// TIA Portal V16 export
// export: Created 2021-11-12T13:31:11.1513233Z, ExportSetting WithDefaults, DisplayName Totally Integrated Automation Portal, DisplayVersion V16 Update 3, DisplayName TIA Portal Version Control Interface, DisplayVersion V16 Update 2, DisplayName TIA Portal Openness, DisplayVersion V16 Update 3, DisplayName SINAMICS Startdrive Advanced, DisplayVersion V16 Update 5, DisplayName SINAMICS Startdrive G130, G150, S120, S150, SINAMICS MV, S210, DisplayVersion V16 Update 5, DisplayName SINAMICS Startdrive G110M, G120, G120C, G120D, G120P, G115D, DisplayVersion V16 Update 5, DisplayName STEP 7 Professional, DisplayVersion V16 Update 3, DisplayName STEP 7 Safety, DisplayVersion V16, DisplayName WinCC UA Professional, DisplayVersion V16 Update 3
DATA_BLOCK "IDB_Sfty_Input"   // DB181, F_DB
{ DB_Accessible_From_OPC_UA := 'FALSE' }
VERSION : 0.1
// stored: AutoNumber true, DBAccessibleFromOPCUA false, InstanceOfName Sfty_Input, InstanceOfType FB
"Sfty_Input"
   // VAR
   //    SF_KAS1 { S7_SetPoint := 'True'} : ESTOP1;
   //    SF_KAS2 { S7_SetPoint := 'True'} : ESTOP1;
   //    SF_BSN1_2 { S7_SetPoint := 'True'} : ESTOP1;
   //    SF_SCH1 { S7_SetPoint := 'True'} : ESTOP1;
   //    SF_BSN3 { S7_SetPoint := 'True'} : ESTOP1;
   //    SF_BSN4_5 { S7_SetPoint := 'True'} : ESTOP1;
   //    SF_THM1 { S7_SetPoint := 'True'} : ESTOP1;
   //    SF_THM2 { S7_SetPoint := 'True'} : ESTOP1;
   //    "SF_1R1-RC01" { S7_SetPoint := 'True'} : ESTOP1;
   //    "SF_1R2-RC01" { S7_SetPoint := 'True'} : ESTOP1;
   //    "SF_1R3-RC01" { S7_SetPoint := 'True'} : ESTOP1;
   //    "SF_1R4-RC01" { S7_SetPoint := 'True'} : ESTOP1;
   //    "SF_1R5-RC01" { S7_SetPoint := 'True'} : ESTOP1;
   //    "SF_1R6-RC01" { S7_SetPoint := 'True'} : ESTOP1;
   //    "SF_2R1-RC01" { S7_SetPoint := 'True'} : ESTOP1;
   //    "SF_2R2-RC01" { S7_SetPoint := 'True'} : ESTOP1;
   //    "SF_000UH11-SF01_12" { S7_SetPoint := 'True'} : ESTOP1;
   //    "SF_000UH10-SF01_12" { S7_SetPoint := 'True'} : ESTOP1;
   //    "SF_100UH11-SF01_12" { S7_SetPoint := 'True'} : ESTOP1;
   //    "SF_100UH12-SF01_12" { S7_SetPoint := 'True'} : ESTOP1;
   //    "SF_100UH13-SF01_12" { S7_SetPoint := 'True'} : ESTOP1;
   //    "SF_100UF01-SF01_12" { S7_SetPoint := 'True'} : ESTOP1;
   //    "SF_200UH11-SF01_12" { S7_SetPoint := 'True'} : ESTOP1;
   //    "SF_200UF01-SF01_12" { S7_SetPoint := 'True'} : ESTOP1;
   //    "SF_210UF01-SF01_12" { S7_SetPoint := 'True'} : ESTOP1;
   //    "SF_220UF01-SF01_12" { S7_SetPoint := 'True'} : ESTOP1;
   //    "SF_230UF01-SF01_12" { S7_SetPoint := 'True'} : ESTOP1;
   //    "SF_300UH11-SF01_12" { S7_SetPoint := 'True'} : ESTOP1;
   //    "SF_310UH31-SF01_12" { S7_SetPoint := 'True'} : ESTOP1;
   //    "SF_330UF01-SF01_12" { S7_SetPoint := 'True'} : ESTOP1;
   //    "SF_400UH11-SF01_12" { S7_SetPoint := 'True'} : ESTOP1;
   //    "SF_400UH31-SF01_12" { S7_SetPoint := 'True'} : ESTOP1;
   //    "SF_410UH31-SF01_12" { S7_SetPoint := 'True'} : ESTOP1;
   //    "SF_420UH31-SF01_12" { S7_SetPoint := 'True'} : ESTOP1;
   //    "SF_100+RU01-QQ01" { S7_SetPoint := 'True'} : ESTOP1;
   //    "SF_100+RU01-QQ02" { S7_SetPoint := 'True'} : ESTOP1;
   //    "SF_100+RU01-QQ03" { S7_SetPoint := 'True'} : ESTOP1;
   //    "SF_100+RU01-QQ04" { S7_SetPoint := 'True'} : ESTOP1;
   //    "SF_100+RU01-QQ05" { S7_SetPoint := 'True'} : ESTOP1;
   //    "SF_100+RU01-QQ06" { S7_SetPoint := 'True'} : ESTOP1;
   //    "SF_100+RU01-QQ07" { S7_SetPoint := 'True'} : ESTOP1;
   //    "SF_100+RU01-QQ08" { S7_SetPoint := 'True'} : ESTOP1;
   //    "SF_200RU01-QQ01" { S7_SetPoint := 'True'} : ESTOP1;
   //    "SF_200RU01-QQ02" { S7_SetPoint := 'True'} : ESTOP1;
   //    "SF_200RU01-QQ03" { S7_SetPoint := 'True'} : ESTOP1;
   //    "SF_200RU01-QQ04" { S7_SetPoint := 'True'} : ESTOP1;
   //    "SF_200RU01-QQ05" { S7_SetPoint := 'True'} : ESTOP1;
   //    "SF_100+RU01-QQ01_lock" { S7_SetPoint := 'True'} : ESTOP1;
   //    "SF_100+RU01-QQ02_lock" { S7_SetPoint := 'True'} : ESTOP1;
   //    "SF_100+RU01-QQ03_lock" { S7_SetPoint := 'True'} : ESTOP1;
   //    "SF_100+RU01-QQ04_lock" { S7_SetPoint := 'True'} : ESTOP1;
   //    "SF_100+RU01-QQ05_lock" { S7_SetPoint := 'True'} : ESTOP1;
   //    "SF_100+RU01-QQ06_lock" { S7_SetPoint := 'True'} : ESTOP1;
   //    "SF_100+RU01-QQ07_lock" { S7_SetPoint := 'True'} : ESTOP1;
   //    "SF_100+RU01-QQ08_lock" { S7_SetPoint := 'True'} : ESTOP1;
   //    "SF_200RU01-QQ01_lock" { S7_SetPoint := 'True'} : ESTOP1;
   //    "SF_200RU01-QQ02_lock" { S7_SetPoint := 'True'} : ESTOP1;
   //    "SF_200RU01-QQ03_lock" { S7_SetPoint := 'True'} : ESTOP1;
   //    "SF_200RU01-QQ04_lock" { S7_SetPoint := 'True'} : ESTOP1;
   //    "SF_200RU01-QQ05_lock" { S7_SetPoint := 'True'} : ESTOP1;
   //    "SF_100+RU01-BG01_close" { S7_SetPoint := 'True'} : ESTOP1;
   //    "SF_100+RU01-BG02_close" { S7_SetPoint := 'True'} : ESTOP1;
   //    "SF_200RU01-BG01_close" { S7_SetPoint := 'True'} : ESTOP1;
   //    "SF_100UR01-KG01R" { S7_SetPoint := 'True'} : ESTOP1;
   //    "SF_100UR01-KG02R" { S7_SetPoint := 'True'} : ESTOP1;
   // END_VAR
BEGIN
END_DATA_BLOCK
